// TIA Portal V15.1 export
// export: Created 2020-06-12T07:35:41.7099609Z, ExportSetting None, DisplayName Totally Integrated Automation Portal, DisplayVersion V15.1, DisplayName TIA Portal Openness, DisplayVersion V15.1, DisplayName STEP 7 Professional, DisplayVersion V15.1, DisplayName STEP 7 Safety, DisplayVersion V15.1, DisplayName WinCC Advanced, DisplayVersion V15.1
FUNCTION "Flags" : Void   // FC10, FBD
TITLE = General program functions / Allgemeine Prog. Funktionen
{ S7_Optimized_Access := 'TRUE' }
AUTHOR : atec
FAMILY : COMMON
NAME : Flags
VERSION : 1.0
// stored: AutoNumber false, SetENOAutomatically False
   VAR_TEMP   // added for the SCL form of the ladder/FBD networks
      _w1 : Bool;
   END_VAR
BEGIN

REGION Network 1: 1 seconds impulse / 1 Sekunden Impuls
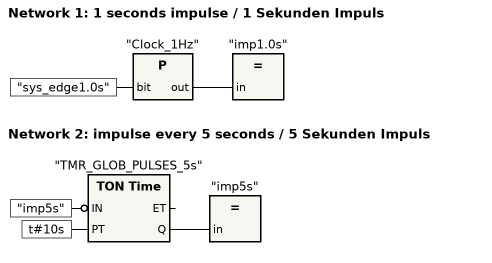
   #_w1 := "Clock_1Hz" AND NOT "sys_edge1.0s";   // rising edge of "Clock_1Hz"
   "sys_edge1.0s" := "Clock_1Hz";
   "imp1.0s" := #_w1;
END_REGION

REGION Network 2: impulse every 5 seconds / 5 Sekunden Impuls
   "TMR_GLOB_PULSES_5s".TON(IN := NOT "imp5s", PT := t#10s);
   "imp5s" := "TMR_GLOB_PULSES_5s".Q;
END_REGION
END_FUNCTION
